Fanuc KAREL source: kt00303.KL

-- PROVISIONAL review KL for V770-1; original PC SHA256 7e43c99f727f0c8103f2d63502856da97d14ab866e82f4a436bdf60fcae79985
-- Incomplete behavior may be omitted. Consult companion uncertainty JSON. Do not deploy.
PROGRAM KT00303
%NOLOCKGROUP
VAR
  I2 : INTEGER
  OUT : BOOLEAN
-- UNRESOLVED_DECL Y1 type=002018
BEGIN
  -- UNRESOLVED_PC offsets 5-19; opcodes 2E,22,9D,33,B2
  -- UNRESOLVED_PC offsets 24-35; opcodes 2E,23
  -- UNRESOLVED_PC offsets 40-62; opcodes 22,9D,33,B1,21,58,23
  -- UNRESOLVED_PC offsets 67-71; opcodes 7F
END KT00303
